TYPE ZDataCalibration :
STRUCT
{region "Handling"}
{IF NOT (defined (Handling_disabled))}
  Handling : HandlingDataCalibration;
  {attribute 'ZId' := 'a0dd13f9-743a-4c3b-9b43-ecc916834d10'}
{END_IF}
{endregion}
{region "Mover1"}
{IF NOT (defined (Mover1_disabled))}
  Mover1 : MoverDataCalibration;
  {attribute 'ZId' := '0635b537-20e6-40de-ab4b-39921311b510'}
{END_IF}
{endregion}
{attribute '__ZwPlcApplicationDataCalibrationDeclaration__'} // Do not remove this attribute! It is used for code generation.
END_STRUCT
END_TYPE

(* stored: Version 1.1.0.1
   DUT ZDataCalibration: Id {a523a901-91d4-4820-87df-fcbb2a68cd13} *)
